Fanuc KAREL source: KT00476.KL

PROGRAM KT00476
%NOLOCKGROUP
VAR
  P1: POSITION
  P2: POSITION
  OUT: XYZWPREXT
BEGIN
  OUT = P1 : P2
END KT00476
